Fanuc KAREL source: kd00067.KL

-- PROVISIONAL review KL for V770-1; original PC SHA256 139d5e5cca894050ebf37fec6ed97ff2e08213cf1a8c24ee515cf4d943674dd7
-- Incomplete behavior may be omitted. Consult companion uncertainty JSON. Do not deploy.
PROGRAM KD00067
%NOLOCKGROUP
VAR
  I : INTEGER
  J : INTEGER
  B : BOOLEAN
  R : REAL
  S : STRING[80]
BEGIN
  -- UNRESOLVED_PC offsets 5-18; opcodes 9D,81,18,9D,1B,9D,12,9C,13,04
  -- UNRESOLVED_PC offsets 23-27; opcodes 7F
END KD00067
